TYPE "UDT_HMI_Alarm_V2"
VERSION : 0.1
   STRUCT
      t : Struct
         x0 : Bool;
         x1 : Bool;
         x2 : Bool;
         x3 : Bool;
         x4 : Bool;
         x5 : Bool;
         x6 : Bool;
         x7 : Bool;
         x8 : Bool;
         x9 : Bool;
         x10 : Bool;
         x11 : Bool;
         x12 : Bool;
         x13 : Bool;
         x14 : Bool;
         x15 : Bool;
      END_STRUCT;
      iHmiSumAlm : Word;
   END_STRUCT;

END_TYPE

TYPE "UDT_PopUp_Allarm"
VERSION : 0.1
   STRUCT
      tEmergencyAlarm { ExternalWritable := 'False'} : Array["STARTARRAY".."DALARM"] of "UDT_HMI_Alarm_V2";
      tAlarm { ExternalWritable := 'False'} : Array["STARTARRAY".."DALARM"] of "UDT_HMI_Alarm_V2";
      tWarning { ExternalWritable := 'False'} : Array["STARTARRAY".."DALARM"] of "UDT_HMI_Alarm_V2";
   END_STRUCT;

END_TYPE

TYPE "UDT_PopUp_Hmi"
VERSION : 0.1
   STRUCT
      tHMR : Struct   // {[Unit]|[Scada Unit]|[LowLimit]|[HigLimit]|[Acces]}
         xManualCommandEnabled { ExternalWritable := 'False'} : Bool;   // Manual Mode Enable {x|x|x|x|O}
         xCleaningEnabled { ExternalWritable := 'False'} : Bool;   // Cleaning Enabled {x|x|x|x|O}
         FrameDown { ExternalWritable := 'False'} : Bool;   // Frame Down {x|x|x|x|O}
         FrameHigh { ExternalWritable := 'False'} : Bool;   // Frame high {x|x|x|x|O}
         PlatePtresence { ExternalWritable := 'False'} : Bool;   // Plate Present {x|x|x|x|O}
         iState { ExternalWritable := 'False'} : Int;   // State PopUp(1=No anomaly, 3=Run, 7=Anomaly) {x|x|x|x|O}
         tManCmd { ExternalWritable := 'False'} : Struct
            xCmdRise { ExternalWritable := 'False'} : Bool;   // Manual Command Rise{x|x|x|x|O}
            xCmdDescend { ExternalWritable := 'False'} : Bool;   // Manual Command Descend{x|x|x|x|O}
         END_STRUCT;
      END_STRUCT;
      tHMW : Struct   // {[Unit]|[Scada Unit]|[LowLimit]|[HigLimit]|[Acces]}
         xStopLocalCleaningRequest : Bool;   // Stop Cleaning {x|x|x|x|O}
         xLocalCleaningRequest : Bool;   // Cleaning Request {x|x|x|x|O}
         xEnableDisableManualCommand : Bool;   // Enable/Disable manual command{x|x|x|x|O}
         tManCmd : Struct
            xCmdRise : Bool;   // Manual Command Rise {x|x|x|x|O}
            xCmdDescend : Bool;   // Manual Command Descend{x|x|x|x|O}
         END_STRUCT;
      END_STRUCT;
   END_STRUCT;

END_TYPE

DATA_BLOCK "PopUp_Alm"
{ S7_Optimized_Access := 'FALSE' }
VERSION : 0.1
NON_RETAIN
   STRUCT
      PopUp : Array["STARTARRAY".."DNUMPOPUP"] of "UDT_PopUp_Allarm";
   END_STRUCT;


BEGIN

END_DATA_BLOCK

DATA_BLOCK "PopUp_Hmi"
{ S7_Optimized_Access := 'FALSE' }
VERSION : 0.1
   STRUCT
      PopUp : Array["STARTARRAY".."DNUMPOPUP"] of "UDT_PopUp_Hmi";
   END_STRUCT;


BEGIN

END_DATA_BLOCK

